DEVICE_TYPE ImageDev (* Device Type *)
  (* Standard: 61499-2 *)
  (* Version 0.0, 2006-01-11, Anirudha, UoA, Added Length and Height *)
  (* Compiler header: package fb.rt.vhmi; import fb.rt.events.*; *)
  VAR_INPUT
    Length : INT;
    Height : INT;
  END_VAR
  RESOURCE_TYPES
    ImageResourceVV;
  END_RESOURCE_TYPES
END_DEVICE_TYPE
